// TIA Portal V16 export
// export: Created 2024-09-05T17:36:34.1141348Z, ExportSetting WithDefaults, DisplayName Totally Integrated Automation Portal, DisplayVersion V16 Update 6, DisplayName TIA Portal Version Control Interface, DisplayVersion V16 Update 2, DisplayName TIA Portal Openness, DisplayVersion V16 Update 6, DisplayName STEP 7 Professional, DisplayVersion V16 Update 6, DisplayName STEP 7 Safety, DisplayVersion V16, DisplayName WinCC Advanced, DisplayVersion V16 Update 6
VAR_GLOBAL   // PLC tag table "Turn table"
   iTurnTableInputs AT %IW300 : Word;
   qTurnTableOutputs AT %QW300 : Word;
   iTurnTableOperating AT %I300.4 : Bool;
   iTurnTableIndexerInPosition AT %I300.5 : Bool;
   qTurnTableStop AT %Q300.1 : Bool;
   qTurnTableCycleCW AT %Q300.2 : Bool;
   qTurnTableCycleCCW AT %Q300.3 : Bool;
   qTurnTableCycleJogCW AT %Q300.4 : Bool;
   qTurnTableCycleJogCCW AT %Q300.5 : Bool;
END_VAR
